// TIA Portal V17 export
// export: Created 2025-05-06T14:45:53.6795227Z, ExportSetting WithDefaults, DisplayName Totally Integrated Automation Portal, DisplayVersion V17 Update 8, DisplayName TIA Portal Openness, DisplayVersion V17 Update 8, DisplayName TIA Portal Version Control Interface, DisplayVersion V17, DisplayName SINAMICS Startdrive Advanced, DisplayVersion V17 SP2, DisplayName SINAMICS Startdrive G110M, G120, G120C, G120D, G120P, G115D, DisplayVersion V17 SP2, DisplayName SINAMICS Startdrive G130, G150, S120, S150, SINAMICS MV, S210, DisplayVersion V17 SP2, DisplayName STEP 7 Professional, DisplayVersion V17 Update 8, DisplayName SINUMERIK ONE STEP 7 Toolbox, DisplayVersion V17 Update 12, DisplayName SINUMERIK 840D sl STEP 7 Toolbox, DisplayVersion V17 Update 12, DisplayName STEP 7 Safety, DisplayVersion V17 Update 6, DisplayName WinCC Advanced, DisplayVersion V17 Update 8
DATA_BLOCK "DB16701_OPC_UA_MASTER_POWDER_2"   // DB16702
{ S7_Optimized_Access := 'FALSE' }
VERSION : 0.1
// stored: AutoNumber false, DBAccessibleFromOPCUA true, DBAccessibleFromWebserver true, IsOnlyStoredInLoadMemory false, IsWriteProtectedInAS false
   VAR RETAIN
      GENERAL : Struct
         ID : Struct
            LINE : Int;   // Line ID
            MACHINE : Int;   // Machine ID
            PLC : Int;   // PLC ID
         END_STRUCT;
         "VERSION" : Struct
            MAJOR : Byte := 0;   // Major version
            MINOR : Byte := 1;   // Minor version
         END_STRUCT;
      END_STRUCT;
      PARAMS : Struct
         UNIT_1 : Struct
            SECTION_4_INNER_DIAMETER : Real;   // combiner-splitter tube inner diameter
            SECTION_4_OUTTER_DIAMETER : Real;   // combiner-splitter tube outer diameter
            SECTION_5_INNER_DIAMETER : Real;   // splitter-inyector tube inner diameter
            SECTION_5_OUTTER_DIAMETER : Real;   // splitter-inyector tube outer diameter
            COMBINER_TYPE : Array[1..40] of Char;   // Combiner model reference
            HOPPER_1 : Struct
               SECTION_1_INNER_DIAMETER : UInt;   // manual valve-pinch valve tube inner diameter
               SECTION_1_OUTTER_DIAMETER : UInt;   // manual valve-pinch valve tube outter diameter
               SECTION_2_INNER_DIAMETER : UInt;   // medicoat-hopper tube inner diameter
               SECTION_2_OUTTER_DIAMETER : UInt;   // medicoat-hopper tube outer diameter
               MIN_WEIGHT : Real;   // Minimun Hopper height
               MAX_WEIGHT : Real;   // Maximun Hopper height
               STIRRER_CURR_THRESHOLD : UInt;   // Low powder level current threshold
               DELTA_PRESSURE : Real;   // Pressure difference setpoint beetwen hopper and feeder hopper
               MAX_PRESSURE : Real;   // Maximun hopper pressure setpoint
               STIRRER_TYPE : Array[1..40] of Char;   // Stirrer model reference
               JACKET_TEMPERATURE : Real;   // Jacket temperature setpoint
               STIRRER_SPEED : Real;   // Stirrer speed setpoint
            END_STRUCT;
            HOPPER_2 : Struct
               SECTION_1_INNER_DIAMETER : UInt;   // manual valve-pinch valve tube inner diameter
               SECTION_1_OUTTER_DIAMETER : UInt;   // manual valve-pinch valve tube outter diameter
               SECTION_2_INNER_DIAMETER : UInt;   // medicoat-hopper tube inner diameter
               SECTION_2_OUTTER_DIAMETER : UInt;   // medicoat-hopper tube outer diameter
               MIN_WEIGHT : Real;   // Minimun Hopper height
               MAX_WEIGHT : Real;   // Maximun Hopper height
               STIRRER_CURR_THRESHOLD : UInt;   // Low powder level current threshold
               DELTA_PRESSURE : Real;   // Pressure difference setpoint beetwen hopper and feeder hopper
               MAX_PRESSURE : Real;   // Maximun hopper pressure setpoint
               STIRRER_TYPE : Array[1..40] of Char;   // Stirrer model reference
               JACKET_TEMPERATURE : Real;   // Jacket temperature setpoint
               STIRRER_SPEED : Real;   // Stirrer speed setpoint
            END_STRUCT;
            FEEDER_1 : Struct
               LINE_1 : Struct
                  STIRRER_SPEED : Real;   // Stirrer speed setpoint
                  WARN_STIRRER_CURR_THRESHOLD : UInt;   // Low powder level current threshold for warning
                  ERR_STIRRER_CURR_THRESHOLD : UInt;   // Low powder level current threshold for alarm
                  STIRRER_TYPE : Array[1..40] of Char;   // Stirrer model reference
                  DUMPER_Z : Real;   // height setpoint between cone and dumper
                  DISC : Struct
                     SPEED : Real;   // Disc speed setpoint
                  END_STRUCT;
                  CARRIER_GAS_FLOW : Real;   // Carrier gas flow setpoint
                  JACKET_TEMPERATURE : Real;   // Jacket temperature setpoint
                  IN_POLIAMYDE_HEIGHT : Real;   // height of the polyamide part at powder inlet
                  OUT_POLIAMYDE_HEIGHT : Real;   // height of the polyamide part at powder outlet
                  IN_POLIAMYDE_ANGLE : Real;   // angle of the polyamide part at powder inlet
                  DISC_PATH_WIDTH : Real;   // Disc path width
                  DISC_PATH_DEPTH : Real;   // Disc path depth
                  MEDICOAT_DIAMETER : Real;   // Medicoat section diameter
                  SECTION_3_INNER_DIAMETER : Real;   // medicoat-combiner tube inner diameter
                  SECTION_3_OUTTER_DIAMETER : Real;   // medicoat-combiner tube outer diameter
               END_STRUCT;
               LINE_2 : Struct
                  STIRRER_SPEED : Real;   // Stirrer speed setpoint
                  WARN_STIRRER_CURR_THRESHOLD : UInt;   // Low powder level current threshold for warning
                  ERR_STIRRER_CURR_THRESHOLD : UInt;   // Low powder level current threshold for alarm
                  STIRRER_TYPE : Array[1..40] of Char;   // Stirrer model reference
                  DUMPER_Z : Real;   // height setpoint between cone and dumper
                  DISC : Struct
                     SPEED : Real;   // Disc speed setpoint
                  END_STRUCT;
                  CARRIER_GAS_FLOW : Real;   // Carrier gas flow setpoint
                  JACKET_TEMPERATURE : Real;   // Jacket temperature setpoint
                  IN_POLIAMYDE_HEIGHT : Real;   // height of the polyamide part at powder inlet
                  OUT_POLIAMYDE_HEIGHT : Real;   // height of the polyamide part at powder outlet
                  IN_POLIAMYDE_ANGLE : Real;   // angle of the polyamide part at powder inlet
                  DISC_PATH_WIDTH : Real;   // Disc path width
                  DISC_PATH_DEPTH : Real;   // Disc path depth
                  MEDICOAT_DIAMETER : Real;   // Medicoat section diameter
                  SECTION_3_INNER_DIAMETER : Real;   // medicoat-combiner tube inner diameter
                  SECTION_3_OUTTER_DIAMETER : Real;   // medicoat-combiner tube outer diameter
               END_STRUCT;
            END_STRUCT;
         END_STRUCT;
         UNIT_2 : Struct
            SECTION_4_INNER_DIAMETER : Real;   // combiner-splitter tube inner diameter
            SECTION_4_OUTTER_DIAMETER : Real;   // combiner-splitter tube outer diameter
            SECTION_5_INNER_DIAMETER : Real;   // splitter-inyector tube inner diameter
            SECTION_5_OUTTER_DIAMETER : Real;   // splitter-inyector tube outer diameter
            COMBINER_TYPE : Array[1..40] of Char;   // Combiner model reference
            HOPPER_1 : Struct
               SECTION_1_INNER_DIAMETER : UInt;   // manual valve-pinch valve tube inner diameter
               SECTION_1_OUTTER_DIAMETER : UInt;   // manual valve-pinch valve tube outter diameter
               SECTION_2_INNER_DIAMETER : UInt;   // medicoat-hopper tube inner diameter
               SECTION_2_OUTTER_DIAMETER : UInt;   // medicoat-hopper tube outer diameter
               MIN_WEIGHT : Real;   // Minimun Hopper height
               MAX_WEIGHT : Real;   // Maximun Hopper height
               STIRRER_CURR_THRESHOLD : UInt;   // Low powder level current threshold
               DELTA_PRESSURE : Real;   // Pressure difference setpoint beetwen hopper and feeder hopper
               MAX_PRESSURE : Real;   // Maximun hopper pressure setpoint
               STIRRER_TYPE : Array[1..40] of Char;   // Stirrer model reference
               JACKET_TEMPERATURE : Real;   // Jacket temperature setpoint
               STIRRER_SPEED : Real;   // Stirrer speed setpoint
            END_STRUCT;
            HOPPER_2 : Struct
               SECTION_1_INNER_DIAMETER : UInt;   // manual valve-pinch valve tube inner diameter
               SECTION_1_OUTTER_DIAMETER : UInt;   // manual valve-pinch valve tube outter diameter
               SECTION_2_INNER_DIAMETER : UInt;   // medicoat-hopper tube inner diameter
               SECTION_2_OUTTER_DIAMETER : UInt;   // medicoat-hopper tube outer diameter
               MIN_WEIGHT : Real;   // Minimun Hopper height
               MAX_WEIGHT : Real;   // Maximun Hopper height
               STIRRER_CURR_THRESHOLD : UInt;   // Low powder level current threshold
               DELTA_PRESSURE : Real;   // Pressure difference setpoint beetwen hopper and feeder hopper
               MAX_PRESSURE : Real;   // Maximun hopper pressure setpoint
               STIRRER_TYPE : Array[1..40] of Char;   // Stirrer model reference
               JACKET_TEMPERATURE : Real;   // Jacket temperature setpoint
               STIRRER_SPEED : Real;   // Stirrer speed setpoint
            END_STRUCT;
            HOPPER_3 : Struct
               SECTION_1_INNER_DIAMETER : UInt;   // manual valve-pinch valve tube inner diameter
               SECTION_1_OUTTER_DIAMETER : UInt;   // manual valve-pinch valve tube outter diameter
               SECTION_2_INNER_DIAMETER : UInt;   // medicoat-hopper tube inner diameter
               SECTION_2_OUTTER_DIAMETER : UInt;   // medicoat-hopper tube outer diameter
               MIN_WEIGHT : Real;   // Minimun Hopper height
               MAX_WEIGHT : Real;   // Maximun Hopper height
               STIRRER_CURR_THRESHOLD : UInt;   // Low powder level current threshold
               DELTA_PRESSURE : Real;   // Pressure difference setpoint beetwen hopper and feeder hopper
               MAX_PRESSURE : Real;   // Maximun hopper pressure setpoint
               STIRRER_TYPE : Array[1..40] of Char;   // Stirrer model reference
               JACKET_TEMPERATURE : Real;   // Jacket temperature setpoint
               STIRRER_SPEED : Real;   // Stirrer speed setpoint
            END_STRUCT;
            FEEDER_1 : Struct
               LINE_1 : Struct
                  STIRRER_SPEED : Real;   // Stirrer speed setpoint
                  WARN_STIRRER_CURR_THRESHOLD : UInt;   // Low powder level current threshold for warning
                  ERR_STIRRER_CURR_THRESHOLD : UInt;   // Low powder level current threshold for alarm
                  STIRRER_TYPE : Array[1..40] of Char;   // Stirrer model reference
                  DUMPER_Z : Real;   // height setpoint between cone and dumper
                  DISC : Struct
                     SPEED : Real;   // Disc speed setpoint
                  END_STRUCT;
                  CARRIER_GAS_FLOW : Real;   // Carrier gas flow setpoint
                  JACKET_TEMPERATURE : Real;   // Jacket temperature setpoint
                  IN_POLIAMYDE_HEIGHT : Real;   // height of the polyamide part at powder inlet
                  OUT_POLIAMYDE_HEIGHT : Real;   // height of the polyamide part at powder outlet
                  IN_POLIAMYDE_ANGLE : Real;   // angle of the polyamide part at powder inlet
                  DISC_PATH_WIDTH : Real;   // Disc path width
                  DISC_PATH_DEPTH : Real;   // Disc path depth
                  MEDICOAT_DIAMETER : Real;   // Medicoat section diameter
                  SECTION_3_INNER_DIAMETER : Real;   // medicoat-combiner tube inner diameter
                  SECTION_3_OUTTER_DIAMETER : Real;   // medicoat-combiner tube outer diameter
               END_STRUCT;
               LINE_2 : Struct
                  STIRRER_SPEED : Real;   // Stirrer speed setpoint
                  WARN_STIRRER_CURR_THRESHOLD : UInt;   // Low powder level current threshold for warning
                  ERR_STIRRER_CURR_THRESHOLD : UInt;   // Low powder level current threshold for alarm
                  STIRRER_TYPE : Array[1..40] of Char;   // Stirrer model reference
                  DUMPER_Z : Real;   // height setpoint between cone and dumper
                  DISC : Struct
                     SPEED : Real;   // Disc speed setpoint
                  END_STRUCT;
                  CARRIER_GAS_FLOW : Real;   // Carrier gas flow setpoint
                  JACKET_TEMPERATURE : Real;   // Jacket temperature setpoint
                  IN_POLIAMYDE_HEIGHT : Real;   // height of the polyamide part at powder inlet
                  OUT_POLIAMYDE_HEIGHT : Real;   // height of the polyamide part at powder outlet
                  IN_POLIAMYDE_ANGLE : Real;   // angle of the polyamide part at powder inlet
                  DISC_PATH_WIDTH : Real;   // Disc path width
                  DISC_PATH_DEPTH : Real;   // Disc path depth
                  MEDICOAT_DIAMETER : Real;   // Medicoat section diameter
                  SECTION_3_INNER_DIAMETER : Real;   // medicoat-combiner tube inner diameter
                  SECTION_3_OUTTER_DIAMETER : Real;   // medicoat-combiner tube outer diameter
               END_STRUCT;
            END_STRUCT;
            FEEDER_2 : Struct
               LINE_2 : Struct
                  STIRRER_SPEED : Real;   // Stirrer speed setpoint
                  WARN_STIRRER_CURR_THRESHOLD : UInt;   // Low powder level current threshold for warning
                  ERR_STIRRER_CURR_THRESHOLD : UInt;   // Low powder level current threshold for alarm
                  STIRRER_TYPE : Array[1..40] of Char;   // Stirrer model reference
                  DUMPER_Z : Real;   // height setpoint between cone and dumper
                  DISC : Struct
                     SPEED : Real;   // Disc speed setpoint
                  END_STRUCT;
                  CARRIER_GAS_FLOW : Real;   // Carrier gas flow setpoint
                  JACKET_TEMPERATURE : Real;   // Jacket temperature setpoint
                  IN_POLIAMYDE_HEIGHT : Real;   // height of the polyamide part at powder inlet
                  OUT_POLIAMYDE_HEIGHT : Real;   // height of the polyamide part at powder outlet
                  IN_POLIAMYDE_ANGLE : Real;   // angle of the polyamide part at powder inlet
                  DISC_PATH_WIDTH : Real;   // Disc path width
                  DISC_PATH_DEPTH : Real;   // Disc path depth
                  MEDICOAT_DIAMETER : Real;   // Medicoat section diameter
                  SECTION_3_INNER_DIAMETER : Real;   // medicoat-combiner tube inner diameter
                  SECTION_3_OUTTER_DIAMETER : Real;   // medicoat-combiner tube outer diameter
               END_STRUCT;
            END_STRUCT;
         END_STRUCT;
      END_STRUCT;
      MONITORING : Struct
         HOPPER_DEC : Struct
            DMC : Array[0..63] of Char;   // Last powder DMC at DEC system input
            LAST_DATE : DTL;   // Last fill in date
            WORKER_ID : Int;   // Last fill in Worker ID
         END_STRUCT;
         UNIT_1 : Struct
            HOPPER_1 : Struct
               PRESSURIZE_PROP_GAS_VALVE_F : Int;   // proportional valve opening level
               PRESSURIZE_GAS_VALVE : Bool;   // pressurization valve open
               RELIEF_GAS_VALVE : Bool;   // relief valve open
               HIGH_LEVEL : Bool;   // Powder high level
               LOW_LEVEL : Bool;   // Powder low level
               TOTAL_WEIGHT : Real;   // Hopper total height
               POWDER_WEIGHT : Real;   // Powder height
               UPPER_JACKET_TEMPERATURE : Real;   // upper jacket temperature
               LOWER_JACKET_TEMPERATURE : Real;   // lower jacket temperature
               HOPPER_PRESSURE : Real;   // Hopper pressure
               STIRRER_CURRENT : DInt;   // Stirrer current
               STIRRER_SPEED : DInt;   // Stirrer speed
               TRANSFER_POWDER_VALVE : Bool;   // pinch valve open
               CLEANING_AIR_VALVE : Bool;   // clean valve open
               POWDER_FLOW : Int;   // medicoat signal
            END_STRUCT;
            HOPPER_2 : Struct
               PRESSURIZE_PROP_GAS_VALVE_F : Int;   // proportional valve opening level
               PRESSURIZE_GAS_VALVE : Bool;   // pressurization valve open
               RELIEF_GAS_VALVE : Bool;   // relief valve open
               HIGH_LEVEL : Bool;   // Powder high level
               LOW_LEVEL : Bool;   // Powder low level
               TOTAL_WEIGHT : Real;   // Hopper total height
               POWDER_WEIGHT : Real;   // Powder height
               UPPER_JACKET_TEMPERATURE : Real;   // upper jacket temperature
               LOWER_JACKET_TEMPERATURE : Real;   // lower jacket temperature
               HOPPER_PRESSURE : Real;   // Hopper pressure
               STIRRER_CURRENT : DInt;   // Stirrer current
               STIRRER_SPEED : DInt;   // Stirrer speed
               TRANSFER_POWDER_VALVE : Bool;   // pinch valve open
               CLEANING_AIR_VALVE : Bool;   // clean valve open
               POWDER_FLOW : Int;   // medicoat signal
            END_STRUCT;
            FEEDER_1 : Struct
               WEIGHT : Real;   // Feeder weight
               LINE_1 : Struct
                  HOPPER : Struct
                     PRESSURE : Real;   // Hopper pressure
                     TEMPERATURE : Real;   // Hopper temperature
                     STIRRER_CURRENT : Real;   // Stirrer current
                     STIRRER_SPEED : Real;   // Stirrer speed
                  END_STRUCT;
                  DISC : Struct
                     CURRENT : Real;   // Disc current
                     SPEED : Real;   // Disc Speed
                  END_STRUCT;
                  CARRIER_GAS : Struct
                     PRESSURE : Real;   // Carrier gas pressure
                     FLOW : Real;   // Carrier gas flow
                  END_STRUCT;
                  POWDER_FLOW : Struct
                     LINE_POWDER_FLOW { S7_SetPoint := 'True'} : Array[1..20] of "MEDICOAT_TIME_STAMP";   // medicoat signal
                  END_STRUCT;
               END_STRUCT;
               LINE_2 : Struct
                  HOPPER : Struct
                     PRESSURE : Real;   // Hopper pressure
                     TEMPERATURE : Real;   // Hopper temperature
                     STIRRER_CURRENT : Real;   // Stirrer current
                     STIRRER_SPEED : Real;   // Stirrer speed
                  END_STRUCT;
                  DISC : Struct
                     CURRENT : Real;   // Disc current
                     SPEED : Real;   // Disc Speed
                  END_STRUCT;
                  CARRIER_GAS : Struct
                     PRESSURE : Real;   // Carrier gas pressure
                     FLOW : Real;   // Carrier gas flow
                  END_STRUCT;
                  POWDER_FLOW : Struct
                     LINE_POWDER_FLOW { S7_SetPoint := 'True'} : Array[1..20] of "MEDICOAT_TIME_STAMP";   // medicoat signal
                  END_STRUCT;
               END_STRUCT;
            END_STRUCT;
            FEEDER_NOZZLE_LINE : Struct
               COMBINER_POWDER_FLOW { S7_SetPoint := 'True'} : Array[1..20] of "MEDICOAT_TIME_STAMP";   // medicoat signal
               NOZZLE_POWDER_FLOW { S7_SetPoint := 'True'} : Array[1..20] of "MEDICOAT_TIME_STAMP";   // medicoat signal
            END_STRUCT;
         END_STRUCT;
         UNIT_2 : Struct
            HOPPER_1 : Struct
               PRESSURIZE_PROP_GAS_VALVE_F : Int;   // proportional valve opening level
               PRESSURIZE_GAS_VALVE : Bool;   // pressurization valve open
               RELIEF_GAS_VALVE : Bool;   // relief valve open
               HIGH_LEVEL : Bool;   // Powder high level
               LOW_LEVEL : Bool;   // Powder low level
               TOTAL_WEIGHT : Real;   // Hopper total height
               POWDER_WEIGHT : Real;   // Powder height
               UPPER_JACKET_TEMPERATURE : Real;   // upper jacket temperature
               LOWER_JACKET_TEMPERATURE : Real;   // lower jacket temperature
               HOPPER_PRESSURE : Real;   // Hopper pressure
               STIRRER_CURRENT : DInt;   // Stirrer current
               STIRRER_SPEED : DInt;   // Stirrer speed
               TRANSFER_POWDER_VALVE : Bool;   // pinch valve open
               CLEANING_AIR_VALVE : Bool;   // clean valve open
               POWDER_FLOW : Int;   // medicoat signal
            END_STRUCT;
            HOPPER_2 : Struct
               PRESSURIZE_PROP_GAS_VALVE_F : Int;   // proportional valve opening level
               PRESSURIZE_GAS_VALVE : Bool;   // pressurization valve open
               RELIEF_GAS_VALVE : Bool;   // relief valve open
               HIGH_LEVEL : Bool;   // Powder high level
               LOW_LEVEL : Bool;   // Powder low level
               TOTAL_WEIGHT : Real;   // Hopper total height
               POWDER_WEIGHT : Real;   // Powder height
               UPPER_JACKET_TEMPERATURE : Real;   // upper jacket temperature
               LOWER_JACKET_TEMPERATURE : Real;   // lower jacket temperature
               HOPPER_PRESSURE : Real;   // Hopper pressure
               STIRRER_CURRENT : DInt;   // Stirrer current
               STIRRER_SPEED : DInt;   // Stirrer speed
               TRANSFER_POWDER_VALVE : Bool;   // pinch valve open
               CLEANING_AIR_VALVE : Bool;   // clean valve open
               POWDER_FLOW : Int;   // medicoat signal
            END_STRUCT;
            HOPPER_3 : Struct
               PRESSURIZE_PROP_GAS_VALVE_F : Int;   // proportional valve opening level
               PRESSURIZE_GAS_VALVE : Bool;   // pressurization valve open
               RELIEF_GAS_VALVE : Bool;   // relief valve open
               HIGH_LEVEL : Bool;   // Powder high level
               LOW_LEVEL : Bool;   // Powder low level
               TOTAL_WEIGHT : Real;   // Hopper total height
               POWDER_WEIGHT : Real;   // Powder height
               UPPER_JACKET_TEMPERATURE : Real;   // upper jacket temperature
               LOWER_JACKET_TEMPERATURE : Real;   // lower jacket temperature
               HOPPER_PRESSURE : Real;   // Hopper pressure
               STIRRER_CURRENT : DInt;   // Stirrer current
               STIRRER_SPEED : DInt;   // Stirrer speed
               TRANSFER_POWDER_VALVE : Bool;   // pinch valve open
               CLEANING_AIR_VALVE : Bool;   // clean valve open
               POWDER_FLOW : Int;   // medicoat signal
            END_STRUCT;
            FEEDER_1 : Struct
               WEIGHT : Real;   // Feeder weight
               LINE_1 : Struct
                  HOPPER : Struct
                     PRESSURE : Real;   // Hopper pressure
                     TEMPERATURE : Real;   // Hopper temperature
                     STIRRER_CURRENT : Real;   // Stirrer current
                     STIRRER_SPEED : Real;   // Stirrer speed
                  END_STRUCT;
                  DISC : Struct
                     CURRENT : Real;   // Disc current
                     SPEED : Real;   // Disc Speed
                  END_STRUCT;
                  CARRIER_GAS : Struct
                     PRESSURE : Real;   // Carrier gas pressure
                     FLOW : Real;   // Carrier gas flow
                  END_STRUCT;
                  POWDER_FLOW : Struct
                     LINE_POWDER_FLOW { S7_SetPoint := 'True'} : Array[1..20] of "MEDICOAT_TIME_STAMP";   // medicoat signal
                  END_STRUCT;
               END_STRUCT;
               LINE_2 : Struct
                  HOPPER : Struct
                     PRESSURE : Real;   // Hopper pressure
                     TEMPERATURE : Real;   // Hopper temperature
                     STIRRER_CURRENT : Real;   // Stirrer current
                     STIRRER_SPEED : Real;   // Stirrer speed
                  END_STRUCT;
                  DISC : Struct
                     CURRENT : Real;   // Disc current
                     SPEED : Real;   // Disc Speed
                  END_STRUCT;
                  CARRIER_GAS : Struct
                     PRESSURE : Real;   // Carrier gas pressure
                     FLOW : Real;   // Carrier gas flow
                  END_STRUCT;
                  POWDER_FLOW : Struct
                     LINE_POWDER_FLOW { S7_SetPoint := 'True'} : Array[1..20] of "MEDICOAT_TIME_STAMP";   // medicoat signal
                  END_STRUCT;
               END_STRUCT;
            END_STRUCT;
            FEEDER_2 : Struct
               WEIGHT : Real;   // Feeder weight
               LINE_2 : Struct
                  HOPPER : Struct
                     PRESSURE : Real;   // Hopper pressure
                     TEMPERATURE : Real;   // Hopper temperature
                     STIRRER_CURRENT : Real;   // Stirrer current
                     STIRRER_SPEED : Real;   // Stirrer speed
                  END_STRUCT;
                  DISC : Struct
                     CURRENT : Real;   // Disc current
                     SPEED : Real;   // Disc Speed
                  END_STRUCT;
                  CARRIER_GAS : Struct
                     PRESSURE : Real;   // Carrier gas pressure
                     FLOW : Real;   // Carrier gas flow
                  END_STRUCT;
                  POWDER_FLOW : Struct
                     LINE_POWDER_FLOW { S7_SetPoint := 'True'} : Array[1..20] of "MEDICOAT_TIME_STAMP";   // medicoat signal
                  END_STRUCT;
               END_STRUCT;
            END_STRUCT;
            FEEDER_NOZZLE_LINE : Struct
               COMBINER_POWDER_FLOW { S7_SetPoint := 'True'} : Array[1..20] of "MEDICOAT_TIME_STAMP";   // medicoat signal
               NOZZLE_POWDER_FLOW { S7_SetPoint := 'True'} : Array[1..20] of "MEDICOAT_TIME_STAMP";   // medicoat signal
            END_STRUCT;
         END_STRUCT;
      END_STRUCT;
      STATUS : Struct
         ACK_BUTTON : Bool;   // Boton para apagar la alarma
         UNIT_1 : Struct
            HOPPER_1 : Struct
               LOAD_HOPPER_SEQ : Bool;   // hopper loading sequence on
               LOAD_FEEDER_SEQ : Bool;   // Feeder loading sequence on
               CLEAN_SEQ : Bool;   // Cleaning secuence on
               PRESSURIZED : Bool;   // Pressurization done
            END_STRUCT;
            HOPPER_2 : Struct
               LOAD_HOPPER_SEQ : Bool;   // hopper loading sequence on
               LOAD_FEEDER_SEQ : Bool;   // Feeder loading sequence on
               CLEAN_SEQ : Bool;   // Cleaning secuence on
               PRESSURIZED : Bool;   // Pressurization done
            END_STRUCT;
            FEEDER_1 : Struct
               GLOBAL_STATUS : Int;   // 1- starting 2- stopping 3- running 4- stopped
               FAULTED : Bool;   // Feeder alarm present
               LINE_1 : Struct
                  POWDER_LEVEL_LOW : Bool;   // Hopper line 1 fill in nedded
               END_STRUCT;
               LINE_2 : Struct
                  POWDER_LEVEL_LOW : Bool;   // Hopper line 2 fill in nedded
               END_STRUCT;
            END_STRUCT;
         END_STRUCT;
         UNIT_2 : Struct
            HOPPER_1 : Struct
               LOAD_HOPPER_SEQ : Bool;   // hopper loading sequence on
               LOAD_FEEDER_SEQ : Bool;   // Feeder loading sequence on
               CLEAN_SEQ : Bool;   // Cleaning secuence on
               PRESSURIZED : Bool;   // Pressurization done
            END_STRUCT;
            HOPPER_2 : Struct
               LOAD_HOPPER_SEQ : Bool;   // hopper loading sequence on
               LOAD_FEEDER_SEQ : Bool;   // Feeder loading sequence on
               CLEAN_SEQ : Bool;   // Cleaning secuence on
               PRESSURIZED : Bool;   // Pressurization done
            END_STRUCT;
            HOPPER_3 : Struct
               LOAD_HOPPER_SEQ : Bool;   // hopper loading sequence on
               LOAD_FEEDER_SEQ : Bool;   // Feeder loading sequence on
               CLEAN_SEQ : Bool;   // Cleaning secuence on
               PRESSURIZED : Bool;   // Pressurization done
            END_STRUCT;
            FEEDER_1 : Struct
               GLOBAL_STATUS : Int;   // 1- starting 2- stopping 3- running 4- stopped
               FAULTED : Bool;   // Feeder alarm present
               LINE_1 : Struct
                  POWDER_LEVEL_LOW : Bool;   // Hopper line 1 fill in nedded
               END_STRUCT;
               LINE_2 : Struct
                  POWDER_LEVEL_LOW : Bool;   // Hopper line 2 fill in nedded
               END_STRUCT;
            END_STRUCT;
            FEEDER_2 : Struct
               GLOBAL_STATUS : Int;   // 1- starting 2- stopping 3- running 4- stopped
               FAULTED : Bool;   // Feeder alarm present
               LINE_2 : Struct
                  POWDER_LEVEL_LOW : Bool;   // Hopper line 1 fill in nedded
               END_STRUCT;
            END_STRUCT;
         END_STRUCT;
         PNEUMATIC : Struct
            POWDER_CONTROL : Struct
               ON : Bool;   // pneumatic system is on
               FAULTED : Bool;   // pneumatic system faulted
            END_STRUCT;
         END_STRUCT;
      END_STRUCT;
      MAINTENANCE : Struct
         MAINT_EVENT : Struct
            REPLACEMENT : Bool;   // Replacement declared by worker
            UNIT_1 : Struct
               SECTION4 : Bool;
               SECTION5 : Bool;
               COMBINER_MEDICOAT : Bool;
               NOZZLE_MEDICOAT : Bool;
               HOPPER_1 : Struct
                  ACTION : Bool;
                  MEDICOAT : Bool;
                  PINCHVALVE : Bool;
                  SECTION1 : Bool;
                  SECTION2 : Bool;
                  LOAD_CELL : Bool;
               END_STRUCT;
               HOPPER_2 : Struct
                  ACTION : Bool;
                  MEDICOAT : Bool;
                  PINCHVALVE : Bool;
                  SECTION1 : Bool;
                  SECTION2 : Bool;
                  LOAD_CELL : Bool;
               END_STRUCT;
               FEEDER_1 : Struct
                  CHANGE : Bool;
                  LINE_1 : Struct
                     HOPPER_CHANGE : Bool;
                     SECTION3 : Bool;
                     MEDICOAT : Bool;
                  END_STRUCT;
                  LINE_2 : Struct
                     HOPPER_CHANGE : Bool;
                     SECTION3 : Bool;
                     MEDICOAT : Bool;
                  END_STRUCT;
               END_STRUCT;
            END_STRUCT;
            UNIT_2 : Struct
               SECTION4 : Bool;
               SECTION5 : Bool;
               COMBINER_MEDICOAT : Bool;
               NOZZLE_MEDICOAT : Bool;
               HOPPER_1 : Struct
                  ACTION : Bool;
                  MEDICOAT : Bool;
                  PINCHVALVE : Bool;
                  SECTION1 : Bool;
                  SECTION2 : Bool;
                  LOAD_CELL : Bool;
               END_STRUCT;
               HOPPER_2 : Struct
                  ACTION : Bool;
                  MEDICOAT : Bool;
                  PINCHVALVE : Bool;
                  SECTION1 : Bool;
                  SECTION2 : Bool;
                  LOAD_CELL : Bool;
               END_STRUCT;
               HOPPER_3 : Struct
                  ACTION : Bool;
                  MEDICOAT : Bool;
                  PINCHVALVE : Bool;
                  SECTION1 : Bool;
                  SECTION2 : Bool;
                  LOAD_CELL : Bool;
               END_STRUCT;
               FEEDER_1 : Struct
                  CHANGE : Bool;
                  LINE_1 : Struct
                     HOPPER_CHANGE : Bool;
                     SECTION3 : Bool;
                     MEDICOAT : Bool;
                  END_STRUCT;
                  LINE_2 : Struct
                     HOPPER_CHANGE : Bool;
                     SECTION3 : Bool;
                     MEDICOAT : Bool;
                  END_STRUCT;
               END_STRUCT;
               FEEDER_2 : Struct
                  CHANGE : Bool;
                  LINE_2 : Struct
                     HOPPER_CHANGE : Bool;
                     SECTION3 : Bool;
                     MEDICOAT : Bool;
                  END_STRUCT;
               END_STRUCT;
            END_STRUCT;
         END_STRUCT;
         MAINT_SEQ : Struct
            UNIT_1 : Struct
               POWDER_FLOW : Bool;
               POWDER_FLOW_RESULT : Real;
               COMBINER_MEDICOAT : Bool;
               NOZZLE_MEDICOAT : Bool;
               HOPPER_1 : Struct
                  SEALING : Bool;
                  SEALING_RESULT : Real;
                  TARE : Bool;
                  MEDICOAT : Bool;
               END_STRUCT;
               HOPPER_2 : Struct
                  SEALING : Bool;
                  SEALING_RESULT : Real;
                  TARE : Bool;
                  MEDICOAT : Bool;
               END_STRUCT;
               FEEDER_1 : Struct
                  FLOWMETER : Bool;
                  DISC : Bool;
                  LINE_1 : Struct
                     SEALING : Bool;
                     SEALING_RESULT : Real;
                     MEDICOAT : Bool;
                  END_STRUCT;
                  LINE_2 : Struct
                     SEALING : Bool;
                     SEALING_RESULT : Real;
                     MEDICOAT : Bool;
                  END_STRUCT;
               END_STRUCT;
            END_STRUCT;
            UNIT_2 : Struct
               POWDER_FLOW : Bool;
               POWDER_FLOW_RESULT : Real;
               COMBINER_MEDICOAT : Bool;
               NOZZLE_MEDICOAT : Bool;
               HOPPER_1 : Struct
                  SEALING : Bool;
                  SEALING_RESULT : Real;
                  TARE : Bool;
                  MEDICOAT : Bool;
               END_STRUCT;
               HOPPER_2 : Struct
                  SEALING : Bool;
                  SEALING_RESULT : Real;
                  TARE : Bool;
                  MEDICOAT : Bool;
               END_STRUCT;
               HOPPER_3 : Struct
                  SEALING : Bool;
                  SEALING_RESULT : Real;
                  TARE : Bool;
                  MEDICOAT : Bool;
               END_STRUCT;
               FEEDER_1 : Struct
                  FLOWMETER : Bool;
                  DISC : Bool;
                  LINE_1 : Struct
                     SEALING : Bool;
                     SEALING_RESULT : Real;
                     MEDICOAT : Bool;
                  END_STRUCT;
                  LINE_2 : Struct
                     SEALING : Bool;
                     SEALING_RESULT : Real;
                     MEDICOAT : Bool;
                  END_STRUCT;
               END_STRUCT;
               FEEDER_2 : Struct
                  FLOWMETER : Bool;
                  DISC : Bool;
                  LINE_2 : Struct
                     SEALING : Bool;
                     SEALING_RESULT : Real;
                     MEDICOAT : Bool;
                  END_STRUCT;
               END_STRUCT;
            END_STRUCT;
         END_STRUCT;
      END_STRUCT;
   END_VAR
BEGIN
END_DATA_BLOCK
